INTERFACE I_ErrorElement

METHOD M_GetError
VAR_INPUT
END_VAR
VAR_OUTPUT
	Error : BOOL;
	ErrorID : DINT;
	ErrorMsg : T_MaxString;
END_VAR
END_METHOD

METHOD M_GetName :STRING
VAR_INPUT
END_VAR
END_METHOD

METHOD RegisterAlarm
VAR_INPUT
	Trigger : REFERENCE TO BOOL;
	ID : DINT;
	value :DINT;
	Message : STRING;
	Category : DINT;
END_VAR
END_METHOD

END_INTERFACE

(* stored: Version 1.1.0.1, ProductVersion 3.1.4024.13
   Itf I_ErrorElement: Id {0f828575-e886-4ef7-bd6f-f5e1150ff524}
   Method M_GetError: Id {1e9cbffb-3e4f-458b-a0ed-3acee17a923c}
   Method M_GetName: Id {86508989-de7e-467c-a96f-d9805e02dbfc}
   Method RegisterAlarm: Id {bda0d40e-fd85-48e4-a39b-c51deb1b027e} *)
